{attribute 'GeneratedUsingTerminal: EK1100-0000-0018'}
{attribute addProperty BoxType "EK1100-0000-0018"}
{attribute addProperty Id "Beckhoff_EP6xxxEK1122Beckhoff_EP6xxxEK1122_6713C7161118"}
{attribute addProperty CRC "789095214"}
{attribute addProperty Size "1118"}
TYPE Beckhoff_EP6xxx_2F08A32E EXTENDS EK1100_1FC0878B :
STRUCT
	{attribute addProperty Name "Beckhoff_EP6xxxEK1122"}
	{attribute addProperty PreviousPort "Beckhoff EP6xxx : B"}
	Beckhoff_EP6xxxEK1122 : Beckhoff_EP6xxxEK1122_6713C716;
END_STRUCT
END_TYPE

(* stored: Version 1.2.0.0, ProductVersion 3.1.4024.9
   DUT Beckhoff_EP6xxx_2F08A32E: Id {3de858f4-3037-44fc-8dce-3ce46afe9e14} *)
